// TIA Portal V20 export
TYPE "LER_typeRFIDConfrolNode"
// stored: Access Published
   STRUCT
      commands { ExternalAccessible := 'False'; ExternalVisible := 'False'; ExternalWritable := 'False'} : "LER_typeRFIDCommands";
      monitoring { ExternalAccessible := 'False'; ExternalVisible := 'False'; ExternalWritable := 'False'} : "LER_typeRFIDMonitoring";
   END_STRUCT;
END_TYPE
